FUNCTION_BLOCK ABSTRACT FB_AbstractLogger IMPLEMENTS I_Logger
VAR_INPUT
	eLogLevel:					E_Event;
END_VAR
VAR_OUTPUT
END_VAR
VAR
END_VAR

METHOD PUBLIC M_Log
VAR_INPUT
	stEvent	: ST_Event;
END_VAR
END_METHOD

END_FUNCTION_BLOCK

(* stored: Version 1.1.0.1
   POU FB_AbstractLogger: Id {e1ce12d2-0f5a-084d-22cb-52e1ac20f2a6}, SpecialFunc None
   Method M_Log: Id {cb7d24f5-cc7a-048b-34f7-d4b522fb60d5} *)
